{attribute 'qualified_only'}
VAR_GLOBAL
    CONSTANT
    EC_MAX_SECONDARY :  BYTE := 10;
    MAX_STRING_SIZE : BYTE := 81;
    NUM_70x1_COE_PARAM : BYTE := 6;
    NUM_SUP_70x1 : BYTE := 4;
END_VAR

(* stored: Version 1.1.0.1, ProductVersion 3.1.4022.18
   GVL GVL_COE: Id {9b0d798d-e9c6-4dcc-9bc7-12a6e92aaaa7} *)
